{attribute 'GeneratedUsingTerminal: EK1100-0000-0018'}
{attribute addProperty BoxType "EK1100-0000-0018"}
{attribute addProperty Id "Beckhoff_EP1xxxEK1122Beckhoff_EP1xxxEK1122_42EA15061572"}
{attribute addProperty CRC "3592571125"}
{attribute addProperty Size "1572"}
TYPE Beckhoff_EP1xxx_D62248F5 EXTENDS EK1100_1FC0878B :
STRUCT
	{attribute addProperty Name "Beckhoff_EP1xxxEK1122"}
	{attribute addProperty PreviousPort "Beckhoff EP1xxx : B"}
	Beckhoff_EP1xxxEK1122 : Beckhoff_EP1xxxEK1122_42EA1506;
END_STRUCT
END_TYPE

(* stored: Version 1.2.0.0, ProductVersion 3.1.4024.9
   DUT Beckhoff_EP1xxx_D62248F5: Id {62f65150-e158-4cf1-817d-aed83a592a5a} *)
